INTERFACE I_KeyValueCollectionChangedEvent EXTENDS I_Event

PROPERTY PUBLIC Target : I_KeyValueCollection
GET
END_GET
END_PROPERTY

END_INTERFACE

(* stored: Version 1.1.0.1, ProductVersion 3.1.4024.12
   Itf I_KeyValueCollectionChangedEvent: Id {c148c255-bbee-42e3-a68d-707c03f28bd1}
   Property Target: Id {fe79283e-bd7f-4eb2-89e5-e1268bff964c}
   Get Get: Id {7c198971-30dc-453b-be41-a90d39d1c3b2} *)
